TYPE AdditionalService_Struct_EAP :
UNION
		Value : INT;
		Bits : Bits_CommonBlock;
END_UNION
END_TYPE

(* stored: Version 1.1.0.1, ProductVersion 3.1.4024.2
   DUT AdditionalService_Struct_EAP: Id {e6aafbb5-ae68-4558-bbef-bc585f5d3de2} *)
